{attribute 'linkalways'} 
{attribute 'no_explicit_call' := 'This FB is a CLASS and must be accessed using methods or properties'}
{attribute 'enable_dynamic_creation'}
FUNCTION_BLOCK Node_F_VN_FillContainerExp_LREAL EXTENDS VisionNode
VAR
    ipContainer : _ITcVnContainer;
    fValue : _LREAL(0.0);
    nStartIdx : _ULINT(0);
    nCount : _ULINT(0);
    hrPrev : _HRESULT(S_OK);
    hresult : _HRESULT(S_OK);
END_VAR

METHOD PUBLIC  Clone : I_Node
VAR
    pNode : POINTER TO Node_F_VN_FillContainerExp_LREAL;
END_VAR
pNode := __NEW(Node_F_VN_FillContainerExp_LREAL);
Clone := pNode^;
END_METHOD

METHOD FB_init : BOOL
VAR_INPUT
    bInitRetains : BOOL; // if TRUE, the retain variables are initialized (warm start / cold start)
    bInCopyCode : BOOL;  // if TRUE, the instance afterwards gets moved into the copy code (online change)
END_VAR
AddInput('ipContainer', ipContainer);
AddParameter('fValue', fValue);
AddParameter('nStartIdx', nStartIdx);
AddParameter('nCount', nCount);
AddInput('hrPrev', hrPrev);
AddOutput('ipContainer', ipContainer);
AddOutput('hresult',hresult);
END_METHOD

METHOD PROTECTED OnExecute
hresult.Value := F_VN_FillContainerExp_LREAL(
    ipContainer := ipContainer.Value,
    fValue := fValue.Value,
    nStartIdx := nStartIdx.Value,
    nCount := nCount.Value,
    hrPrev:= hrPrev.Value);
END_METHOD

METHOD PUBLIC PreExecutionCheck
VAR_INPUT
    Check : I_PreExecutionChecks;
END_VAR
Check.IsTrue(ipContainer.IsValid, 'ipContainer must be a valid container');
Check.IsTrue(ipContainer.IsType(TC_GLOBAL_CONST_LIST.ContainerType_Vector_LREAL), 'ipContainer contains incorrect type');
END_METHOD

END_FUNCTION_BLOCK

(* stored: Version 1.1.0.1, ProductVersion 3.1.4026.13
   POU Node_F_VN_FillContainerExp_LREAL: Id {c4e9ade6-8e9f-4e1e-81c1-caa6ac5764bb}, SpecialFunc None
   Folder Constructor: Id {5c224e2a-ac19-46b2-9a45-e996c7f8c5c2}
   Method Clone: Id {22b918e5-cf6a-4012-bf2f-be360b4fb66a}
   Method FB_init: Id {83ecc41e-4043-45b4-a712-c51070493f1f}
   Method OnExecute: Id {a861fcff-550f-4272-9319-621f14312a2a}
   Method PreExecutionCheck: Id {ec695394-1106-4533-ba0f-49406d9c8220} *)
